Fanuc KAREL source: kf00056.KL

-- PROVISIONAL review KL for V1013-1; original PC SHA256 1fcb5fedd88b94b76c39ef85cf3eb501b657d596254bd911b5895d378c7908b1
-- Incomplete behavior may be omitted. Consult companion uncertainty JSON. Do not deploy.
PROGRAM KF00056
%NOLOCKGROUP
VAR
  I : INTEGER
  J : INTEGER
  X : REAL
  Y : REAL
  B : BOOLEAN
  C : BOOLEAN
  TXT : STRING[80]
  TXT2 : STRING[80]
  STATUS : INTEGER
-- UNRESOLVED_DECL AI type=002010
-- UNRESOLVED_DECL BI type=002010
-- UNRESOLVED_DECL P type=000102
-- UNRESOLVED_DECL JP type=000199
-- UNRESOLVED_DECL PF type=000101
-- UNRESOLVED_DECL V1 type=000013
-- UNRESOLVED_DECL V2 type=000013
BEGIN
  -- UNRESOLVED_PC offsets 5-15; opcodes 03,9D,1B,12,13,04,14
  -- UNRESOLVED_PC offsets 20-24; opcodes 7F
END KF00056
